TYPE St_Assy_Complete EXTENDS St_Assy_Base :
STRUCT
	eState		:E_AssyComplete;
END_STRUCT
END_TYPE

(* stored: Version 1.1.0.1
   DUT St_Assy_Complete: Id {834e0b4f-0972-4dd9-ac5e-666f73992e25} *)
